(* Logix 5000 project; controller Transcat_L33ER vendor 1 type 14 code 107 rev 32.11; software revision 32.02; part 3 of 4 *)
(* tags used below, declared in another part *)
   AllDevice1stScanDone : BOOL;   // When this bit is set - all devices have been scanned once and bits reset
   AllDeviceEnable : BOOL;   // A bit to enable or disable the running of all devices
   AllReset : BOOL;   // Bit to reset Auto/Man, AutoRun, RecipeRun, TimedRunEnable to 0 from PLC
   alwaysOFF : BOOL;
   AnyAutoRun : BOOL;   // Bit that in on if ANY device is placed into Auto run (to signal pre-start beed)
   AnyAutoRunFlag : BOOL;   // A flag that indicates if any device is in Auto Run (used with pre-start beep logic)
   AnyManRunFlag : BOOL;   // A flag that indicates if any device is in Manual Run (used with pre-start beep logic)
   AnyManualRun : BOOL;   // Bit that in on if ANY device is placed into manual run (to signal pre-start beed)
   Auto_Run_All_Interlock : BOOL;   // Bit to interlock all devices running in Auto
   AutoActive : BOOL;   // Auto mode active
   Beep : BOOL;   // Bit to Activte Beacon Alarm
   Device : Device[20];
   DiscreteTemp : BOOL;   // A temporay boolean to hold positions during PLC transer
   dNum : DINT;   // The index of the current device being processed
   DoseCounter : COUNTER;   // Counts the # of doses since last reset
   DoseCounterReset_HMI : BOOL;   // HMI bit to reset the dose counter
   DoseStart : BOOL;   // Bit to start dosing sequence
   DoseStartOneShot : BOOL;   // One shot to start dosing
   DoseStop : BOOL;   // Bit to stop dosing
   DoseStopOneShot : BOOL;   // one shot to stop dosing
   DoseTarget : REAL;   // Target dose amount
   EstopActive : BOOL;   // E
   EstopFalutResetTOF : TIMER;   // Timer to hold reset bit to allow all drives to reset
   EStopResetPulse : BOOL;   // One-scan pulse used to clear all 14 E-stop interlocks - allows reset of estop interlocks from physical reset button on V
   EStopResetRequired : BOOL;   // Indicates that an estop was actived and it's awaiting reset
   FT103 : BronkhorstFlowMeter;
   FT103B : BronkhorstFlowMeter;
   GF101 : Thayer_WB_Feeder;   // Thayer 1 Tags
   GF101_Write_Acknowledge : ALIAS FOR Thayer1_BS:O.Data[2].5;   // Thayer 1 (GF101) Acknowledge
   GF201 : Thayer_WB_Feeder;   // Thayer 2 Tags
   GF201_Totalizer1 : ALIAS FOR Thayer2Data[9];   // Thayer 2 (GF201) Totalizer 1 in lbs
   GF201_Write_Acknowledge : ALIAS FOR Thayer2_BS:O.Data[2].5;   // Thayer 2 (GF201) Acknowledge
   GF201_Write_Total1Reset : ALIAS FOR Thayer2_BS:O.Data[2].1;   // Thayer 2 (GF1201) Totalizer 1 reset
   HMI_AllReset : BOOL;   // Bit to reset Auto/Man, AutoRun, RecipeRun, TimedRunEnable to 0 from HMI
   HMI_AutoStart : BOOL;   // Starts all devices in AUTO
   HMI_AutoStop : BOOL;   // Stops all devices in AUTO
   HMI_RecipeStart : BOOL;   // Bit to start and stop recipe from HMI
   InitCount : INT;   // Counter to cycle through each device on start-up and reset AutoMan, AutoRun, ManualRun bits
   MX101 : Howes_Mixer;
   MX201 : Howes_Mixer;
   RecipeStart : BOOL;   // Bit to start and stop a recipe execution from PLC logic
   StartBeepTimer : TIMER;   // Timer to sound the beep alarm before starting a device
   TestBit1 : BOOL;   // Just a test bit - does not do anything
   Thayer2ResetTotal1_HMI : BOOL;   // Bit to reset Thayer2 - totalizer 1 from HMI
   VF101 : Acrison_Feeder;   // Medium Feeder Tags
   VF201 : Acrison_Feeder;   // Small Feeder 2 Tags
   VFD_Panel_Safety_Panel_Etop_OK : ALIAS FOR XS26_VFD_Cabinet_Safety_Controller:I1.Data[1].6;
   VFD_Panel_Safety_Remote_Estops_OK : ALIAS FOR XS26_VFD_Cabinet_Safety_Controller:I1.Data[1].7;
(* MainProgram, continued *)

ROUTINE DeviceLogic   (* ladder *)
// Process the logic for each device with index and indirect addressing.
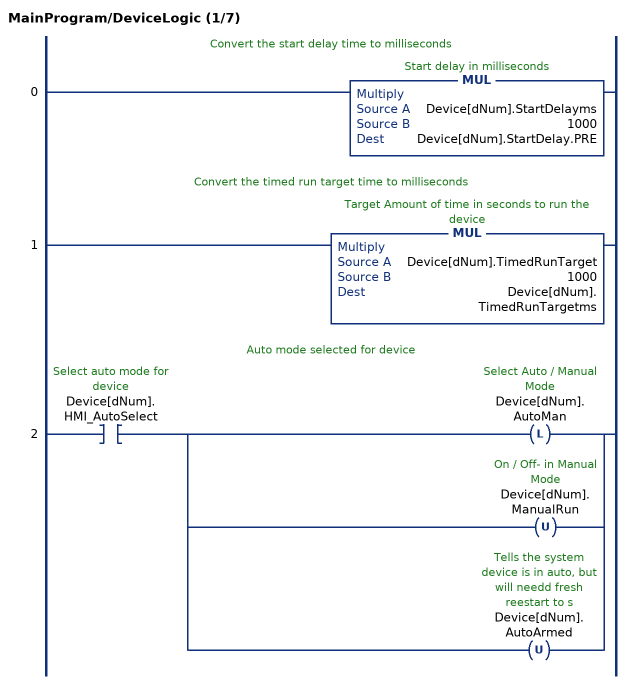
   // Convert the start delay time to milliseconds
   0: MUL(Device[dNum].StartDelayms,1000,Device[dNum].StartDelay.PRE);
   // Convert the timed run target time to milliseconds
   1: MUL(Device[dNum].TimedRunTarget,1000,Device[dNum].TimedRunTargetms);
   // Auto mode selected for device
   2: XIC(Device[dNum].HMI_AutoSelect)[OTL(Device[dNum].AutoMan) ,OTU(Device[dNum].ManualRun) ,OTU(Device[dNum].AutoArmed) ];
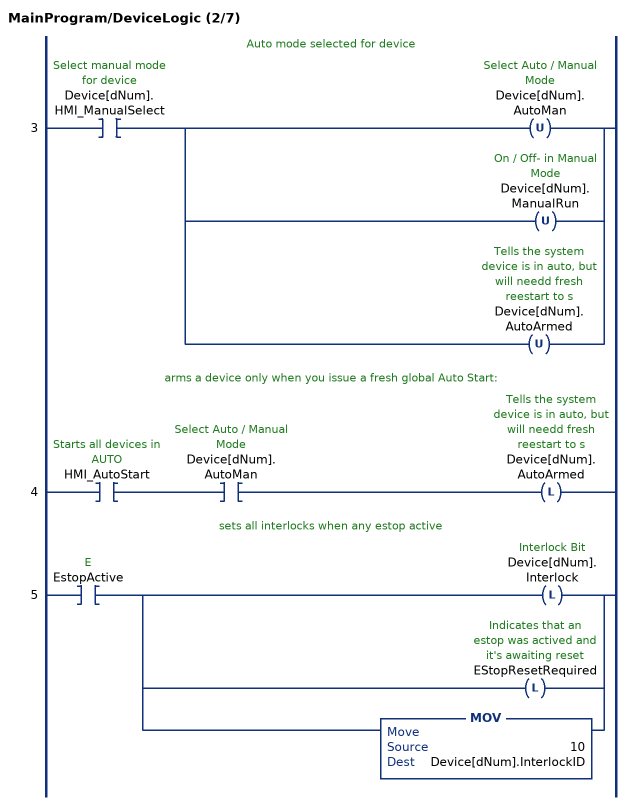
   // Auto mode selected for device
   3: XIC(Device[dNum].HMI_ManualSelect)[OTU(Device[dNum].AutoMan) ,[OTU(Device[dNum].ManualRun) ,OTU(Device[dNum].AutoArmed) ] ];
   // arms a device only when you issue a fresh global Auto Start:
   4: XIC(HMI_AutoStart)XIC(Device[dNum].AutoMan)OTL(Device[dNum].AutoArmed);
   // sets all interlocks when any estop active
   5: XIC(EstopActive)[OTL(Device[dNum].Interlock) ,OTL(EStopResetRequired) ,MOV(10,Device[dNum].InterlockID) ];
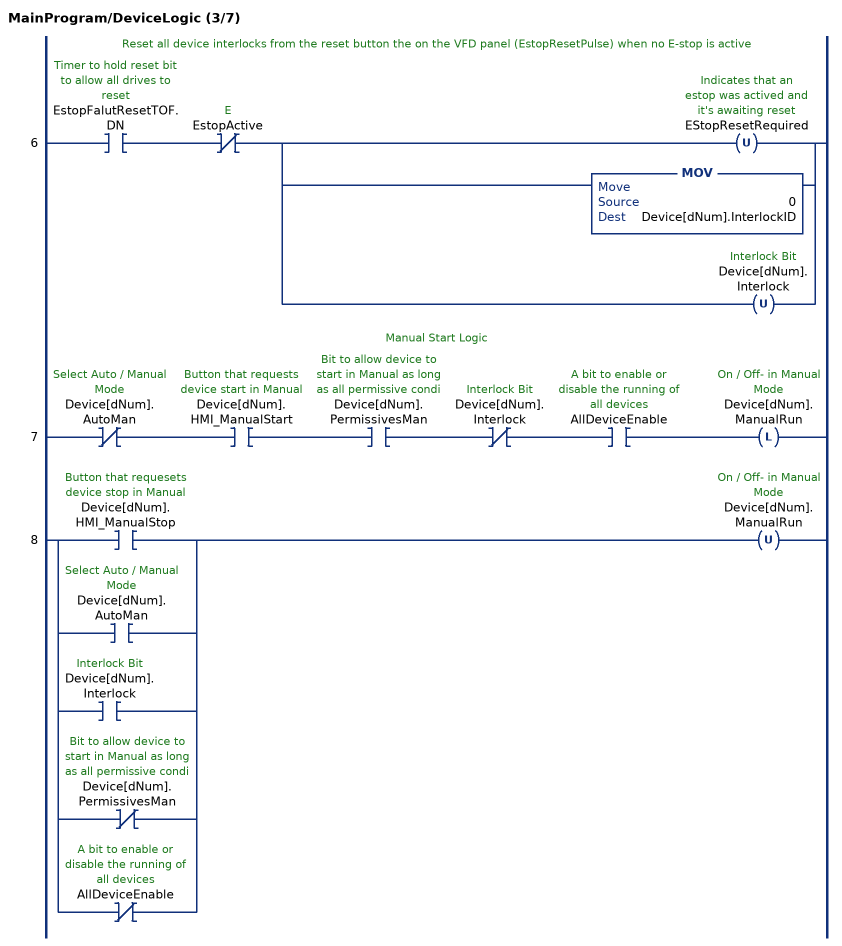
   // Reset all device interlocks from the reset button the on the VFD panel (EstopResetPulse) when no E-stop is active
   6: XIC(EstopFalutResetTOF.DN)XIO(EstopActive)[OTU(EStopResetRequired) ,MOV(0,Device[dNum].InterlockID) ,OTU(Device[dNum].Interlock) ];
   // Manual Start Logic
   7: XIO(Device[dNum].AutoMan)XIC(Device[dNum].HMI_ManualStart)XIC(Device[dNum].PermissivesMan)XIO(Device[dNum].Interlock)XIC(AllDeviceEnable)OTL(Device[dNum].ManualRun);
   8: [XIC(Device[dNum].HMI_ManualStop) ,[XIC(Device[dNum].AutoMan) ,[XIC(Device[dNum].Interlock) ,[XIO(Device[dNum].PermissivesMan) ,XIO(AllDeviceEnable) ] ] ] ]OTU(Device[dNum].ManualRun);
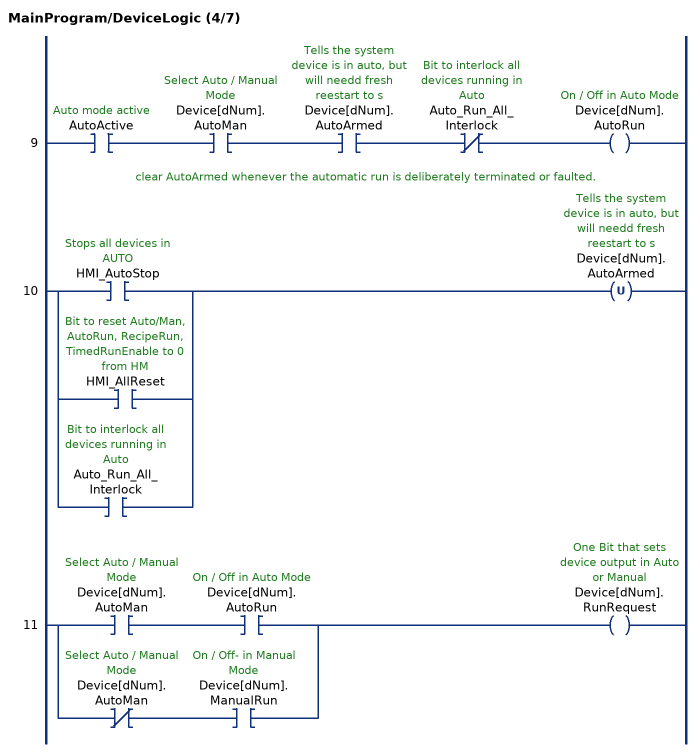
   9: XIC(AutoActive)XIC(Device[dNum].AutoMan)XIC(Device[dNum].AutoArmed)XIO(Auto_Run_All_Interlock)OTE(Device[dNum].AutoRun);
   // clear AutoArmed whenever the automatic run is deliberately terminated or faulted.
   10: [XIC(HMI_AutoStop) ,[XIC(HMI_AllReset) ,XIC(Auto_Run_All_Interlock) ] ]OTU(Device[dNum].AutoArmed);
   11: [XIC(Device[dNum].AutoMan) XIC(Device[dNum].AutoRun) ,XIO(Device[dNum].AutoMan) XIC(Device[dNum].ManualRun) ]OTE(Device[dNum].RunRequest);
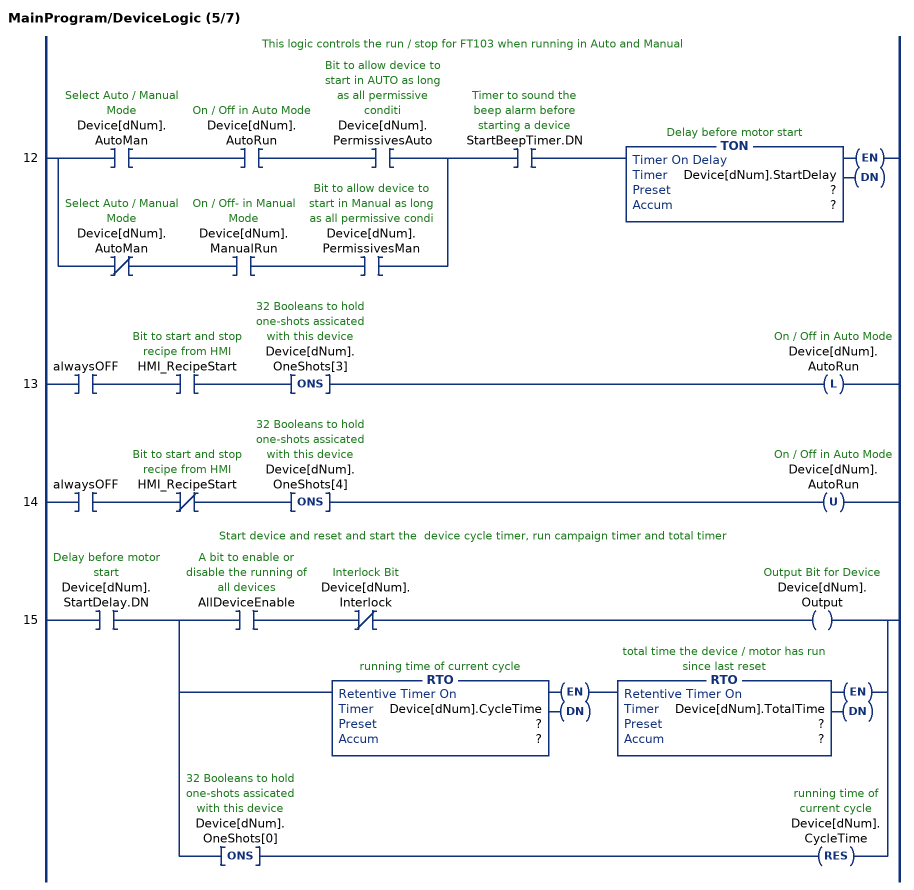
   // This logic controls the run / stop for FT103 when running in Auto and Manual
   12: [XIC(Device[dNum].AutoMan) XIC(Device[dNum].AutoRun) XIC(Device[dNum].PermissivesAuto) ,XIO(Device[dNum].AutoMan) XIC(Device[dNum].ManualRun) XIC(Device[dNum].PermissivesMan) ]XIC(StartBeepTimer.DN)TON(Device[dNum].StartDelay,?,?);
   13: XIC(alwaysOFF)XIC(HMI_RecipeStart)ONS(Device[dNum].OneShots[3])OTL(Device[dNum].AutoRun);
   14: XIC(alwaysOFF)XIO(HMI_RecipeStart)ONS(Device[dNum].OneShots[4])OTU(Device[dNum].AutoRun);
   // Start device and reset and start the  device cycle timer, run campaign timer and total timer
   15: XIC(Device[dNum].StartDelay.DN)[XIC(AllDeviceEnable) XIO(Device[dNum].Interlock) OTE(Device[dNum].Output) ,[RTO(Device[dNum].CycleTime,?,?) RTO(Device[dNum].TotalTime,?,?) ,ONS(Device[dNum].OneShots[0]) RES(Device[dNum].CycleTime) ] ];
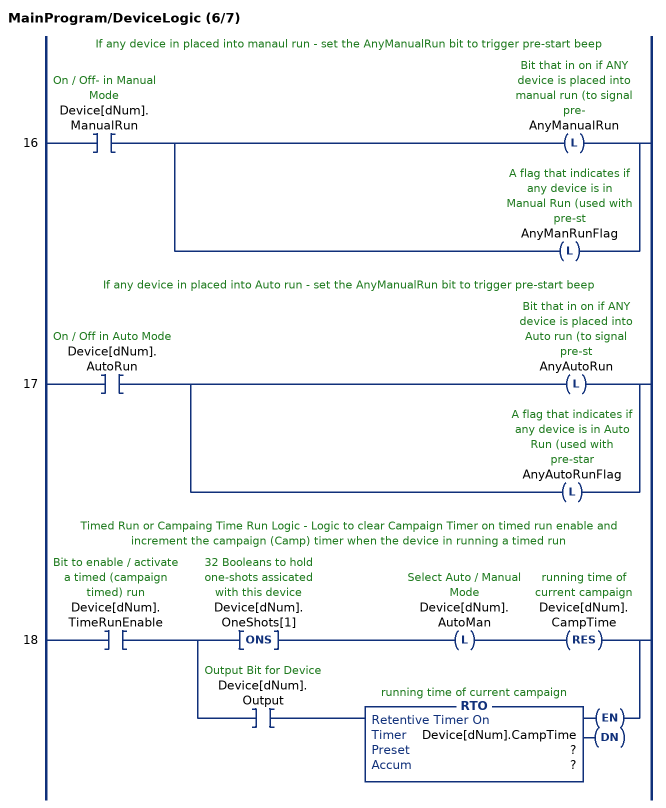
   // If any device in placed into manaul run - set the AnyManualRun bit to trigger pre-start beep
   16: XIC(Device[dNum].ManualRun)[OTL(AnyManualRun) ,OTL(AnyManRunFlag) ];
   // If any device in placed into Auto run - set the AnyManualRun bit to trigger pre-start beep
   17: XIC(Device[dNum].AutoRun)[OTL(AnyAutoRun) ,OTL(AnyAutoRunFlag) ];
   // Timed Run or Campaing Time Run Logic - Logic to clear Campaign Timer on timed run enable and increment the campaign (Camp) timer when the device in running a timed run
   18: XIC(Device[dNum].TimeRunEnable)[ONS(Device[dNum].OneShots[1]) OTL(Device[dNum].AutoMan) RES(Device[dNum].CampTime) ,XIC(Device[dNum].Output) RTO(Device[dNum].CampTime,?,?) ];
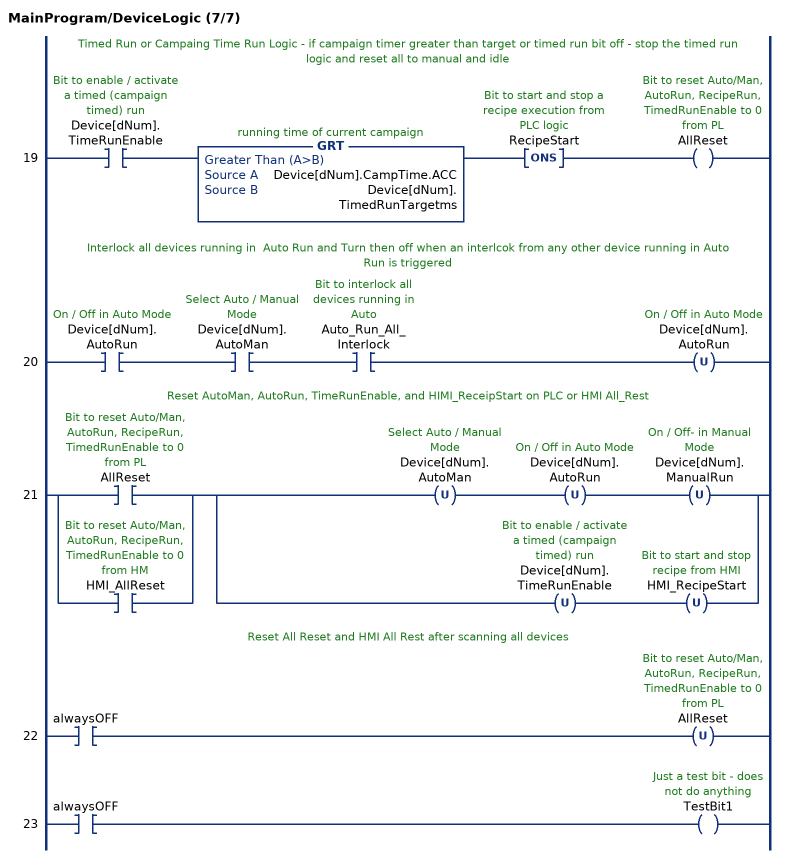
   // Timed Run or Campaing Time Run Logic - if campaign timer greater than target or timed run bit off - stop the timed run logic and reset all to manual and idle
   19: XIC(Device[dNum].TimeRunEnable)GRT(Device[dNum].CampTime.ACC,Device[dNum].TimedRunTargetms)ONS(RecipeStart)OTE(AllReset);
   // Interlock all devices running in  Auto Run and Turn then off when an interlcok from any other device running in Auto Run is triggered
   20: XIC(Device[dNum].AutoRun)XIC(Device[dNum].AutoMan)XIC(Auto_Run_All_Interlock)OTU(Device[dNum].AutoRun);
   // Reset AutoMan, AutoRun, TimeRunEnable, and HIMI_ReceipStart on PLC or HMI All_Rest
   21: [XIC(AllReset) ,XIC(HMI_AllReset) ][OTU(Device[dNum].AutoMan) OTU(Device[dNum].AutoRun) OTU(Device[dNum].ManualRun) ,OTU(Device[dNum].TimeRunEnable) OTU(HMI_RecipeStart) ];
   // Reset All Reset and HMI All Rest after scanning all devices
   22: XIC(alwaysOFF)OTU(AllReset);
   23: XIC(alwaysOFF)OTE(TestBit1);
END_ROUTINE

ROUTINE DeviceManager   (* ladder *)
// Loop through all devices each scan
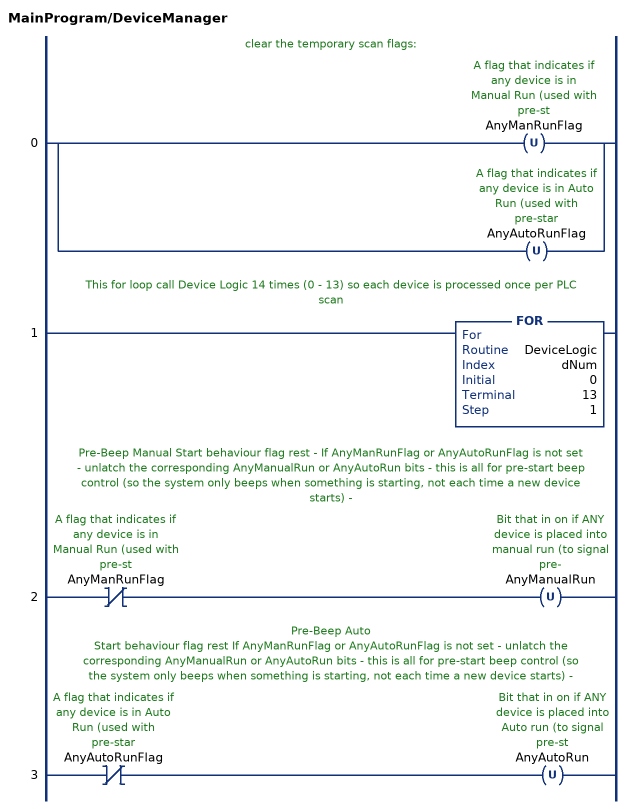
   // clear the temporary scan flags:
   0: [OTU(AnyManRunFlag) ,OTU(AnyAutoRunFlag) ];
   // This for loop call Device Logic 14 times (0 - 13) so each device is processed once per PLC scan
   1: FOR(DeviceLogic,dNum,0,13,1);
   // Pre-Beep Manual Start behaviour flag rest - If AnyManRunFlag or AnyAutoRunFlag is not set - unlatch the corresponding AnyManualRun or AnyAutoRun bits - this is all for pre-start beep control (so the system only beeps when something is starting, not each time a new device starts) -
   2: XIO(AnyManRunFlag)OTU(AnyManualRun);
   // Pre-Beep Auto
   //  Start behaviour flag rest If AnyManRunFlag or AnyAutoRunFlag is not set - unlatch the corresponding AnyManualRun or AnyAutoRun bits - this is all for pre-start beep control (so the system only beeps when something is starting, not each time a new device starts) -
   3: XIO(AnyAutoRunFlag)OTU(AnyAutoRun);
END_ROUTINE

ROUTINE GF201Dose   (* ladder *)
// Logic to Dose a specific amount from GF201 - Thayer 2
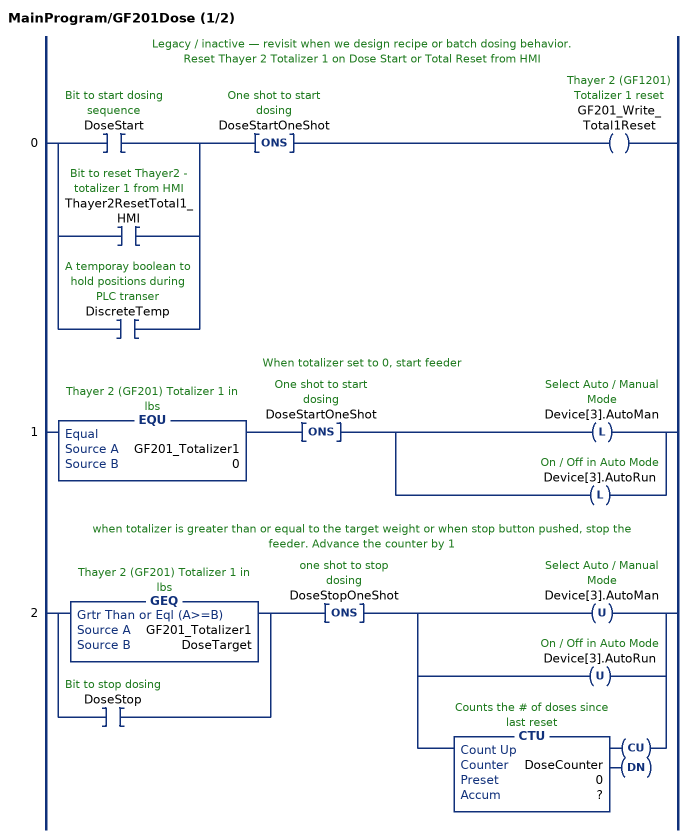
   // Legacy / inactive — revisit when we design recipe or batch dosing behavior.
   // Reset Thayer 2 Totalizer 1 on Dose Start or Total Reset from HMI
   0: [XIC(DoseStart) ,[XIC(Thayer2ResetTotal1_HMI) ,XIC(DiscreteTemp) ] ]ONS(DoseStartOneShot)OTE(GF201_Write_Total1Reset);
   // When totalizer set to 0, start feeder
   1: EQU(GF201_Totalizer1,0)ONS(DoseStartOneShot)[OTL(Device[3].AutoMan) ,OTL(Device[3].AutoRun) ];
   // when totalizer is greater than or equal to the target weight or when stop button pushed, stop the feeder. Advance the counter by 1
   2: [GEQ(GF201_Totalizer1,DoseTarget) ,XIC(DoseStop) ]ONS(DoseStopOneShot)[OTU(Device[3].AutoMan) ,[OTU(Device[3].AutoRun) ,CTU(DoseCounter,?,?) ] ];
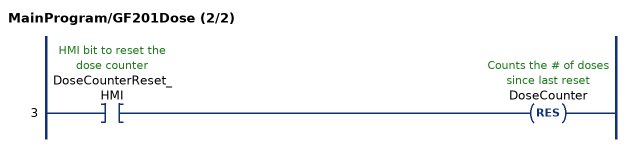
   3: XIC(DoseCounterReset_HMI)RES(DoseCounter);
END_ROUTINE

ROUTINE Initialize   (* ladder *)
// Reset controls and any other initialization required
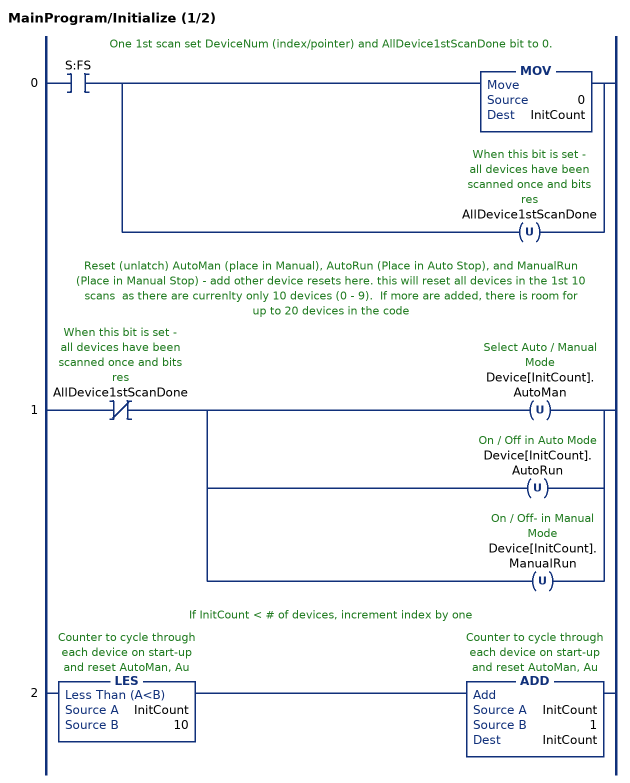
   // One 1st scan set DeviceNum (index/pointer) and AllDevice1stScanDone bit to 0.
   0: XIC(S:FS)[MOV(0,InitCount) ,OTU(AllDevice1stScanDone) ];
   // Reset (unlatch) AutoMan (place in Manual), AutoRun (Place in Auto Stop), and ManualRun (Place in Manual Stop) - add other device resets here. this will reset all devices in the 1st 10 scans  as there are currenlty only 10 devices (0 - 9).  If more are added, there is room for up to 20 devices in the code
   1: XIO(AllDevice1stScanDone)[OTU(Device[InitCount].AutoMan) ,[OTU(Device[InitCount].AutoRun) ,OTU(Device[InitCount].ManualRun) ] ];
   // If InitCount < # of devices, increment index by one
   2: LES(InitCount,10)ADD(InitCount,1,InitCount);
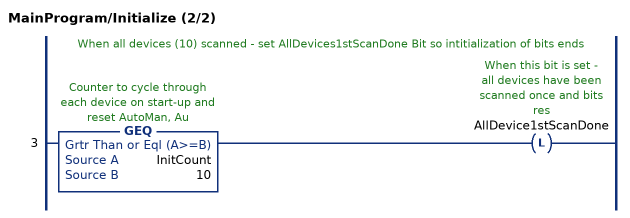
   // When all devices (10) scanned - set AllDevices1stScanDone Bit so intitialization of bits ends
   3: GEQ(InitCount,10)OTL(AllDevice1stScanDone);
END_ROUTINE

ROUTINE InterlockLogic   (* ladder *)
// All interlock logic is handled here
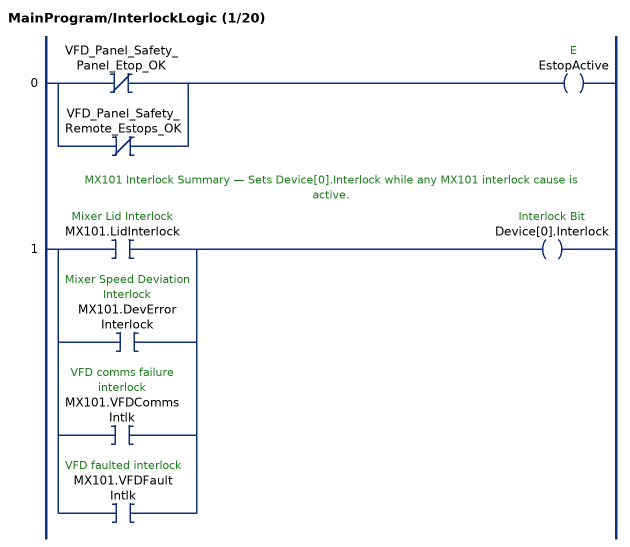
   0: [XIO(VFD_Panel_Safety_Panel_Etop_OK) ,XIO(VFD_Panel_Safety_Remote_Estops_OK) ]OTE(EstopActive);
   // MX101 Interlock Summary — Sets Device[0].Interlock while any MX101 interlock cause is active.
   1: [XIC(MX101.LidInterlock) ,XIC(MX101.DevErrorInterlock) ,XIC(MX101.VFDCommsIntlk) ,XIC(MX101.VFDFaultIntlk) ]OTE(Device[0].Interlock);
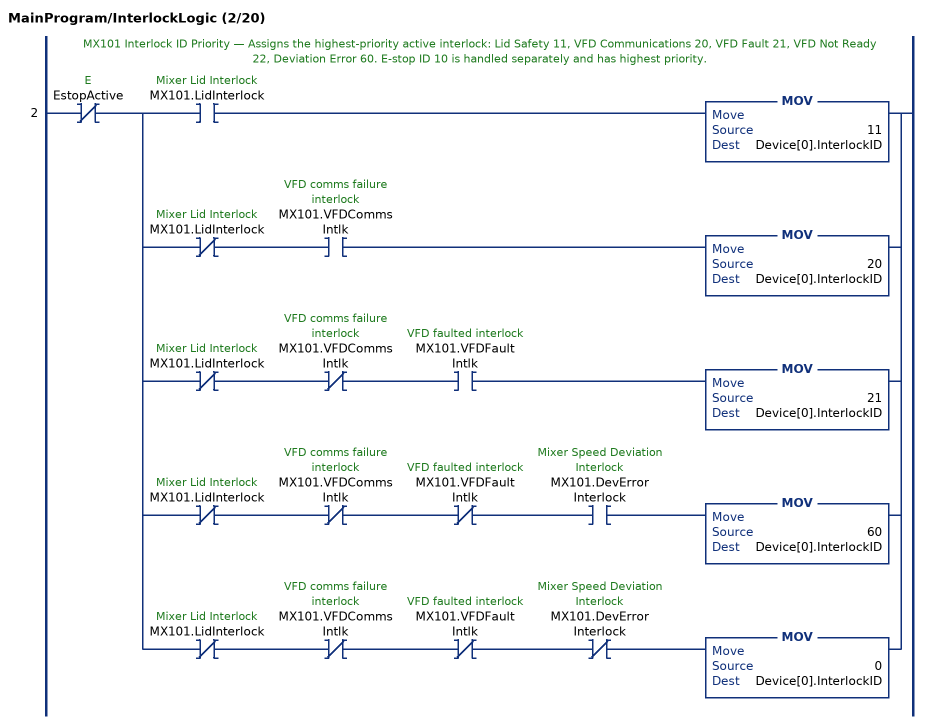
   // MX101 Interlock ID Priority — Assigns the highest-priority active interlock: Lid Safety 11, VFD Communications 20, VFD Fault 21, VFD Not Ready 22, Deviation Error 60. E-stop ID 10 is handled separately and has highest priority.
   2: XIO(EstopActive)[XIC(MX101.LidInterlock) MOV(11,Device[0].InterlockID) ,XIO(MX101.LidInterlock) XIC(MX101.VFDCommsIntlk) MOV(20,Device[0].InterlockID) ,XIO(MX101.LidInterlock) XIO(MX101.VFDCommsIntlk) XIC(MX101.VFDFaultIntlk) MOV(21,Device[0].InterlockID) ,XIO(MX101.LidInterlock) XIO(MX101.VFDCommsIntlk) XIO(MX101.VFDFaultIntlk) XIC(MX101.DevErrorInterlock) MOV(60,Device[0].InterlockID) ,XIO(MX101.LidInterlock) XIO(MX101.VFDCommsIntlk) XIO(MX101.VFDFaultIntlk) XIO(MX101.DevErrorInterlock) MOV(0,Device[0].InterlockID) ];
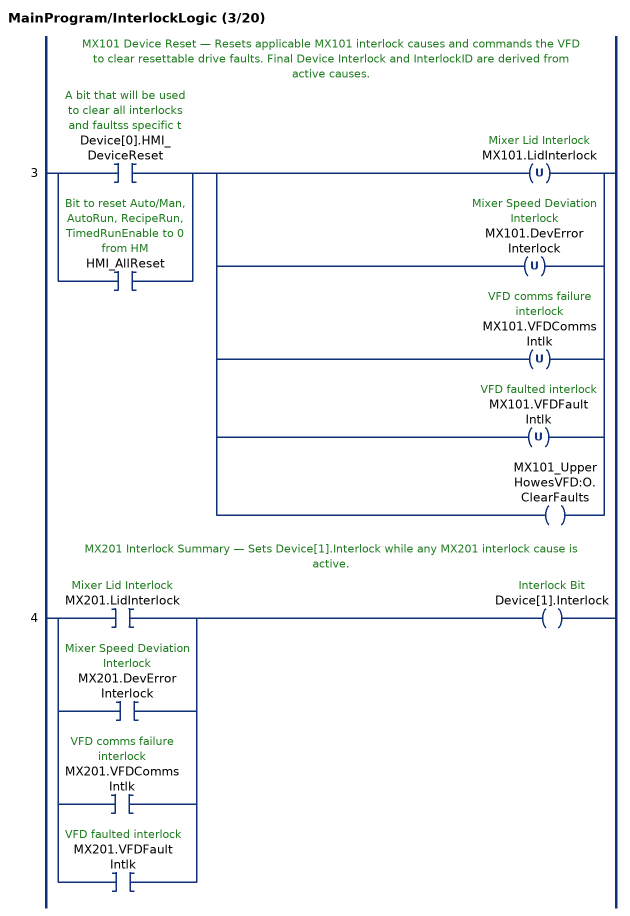
   // MX101 Device Reset — Resets applicable MX101 interlock causes and commands the VFD to clear resettable drive faults. Final Device Interlock and InterlockID are derived from active causes.
   3: [XIC(Device[0].HMI_DeviceReset) ,XIC(HMI_AllReset) ][OTU(MX101.LidInterlock) ,OTU(MX101.DevErrorInterlock) ,OTU(MX101.VFDCommsIntlk) ,OTU(MX101.VFDFaultIntlk) ,OTE(MX101_UpperHowesVFD:O.ClearFaults) ];
   // MX201 Interlock Summary — Sets Device[1].Interlock while any MX201 interlock cause is active.
   4: [XIC(MX201.LidInterlock) ,XIC(MX201.DevErrorInterlock) ,XIC(MX201.VFDCommsIntlk) ,XIC(MX201.VFDFaultIntlk) ]OTE(Device[1].Interlock);
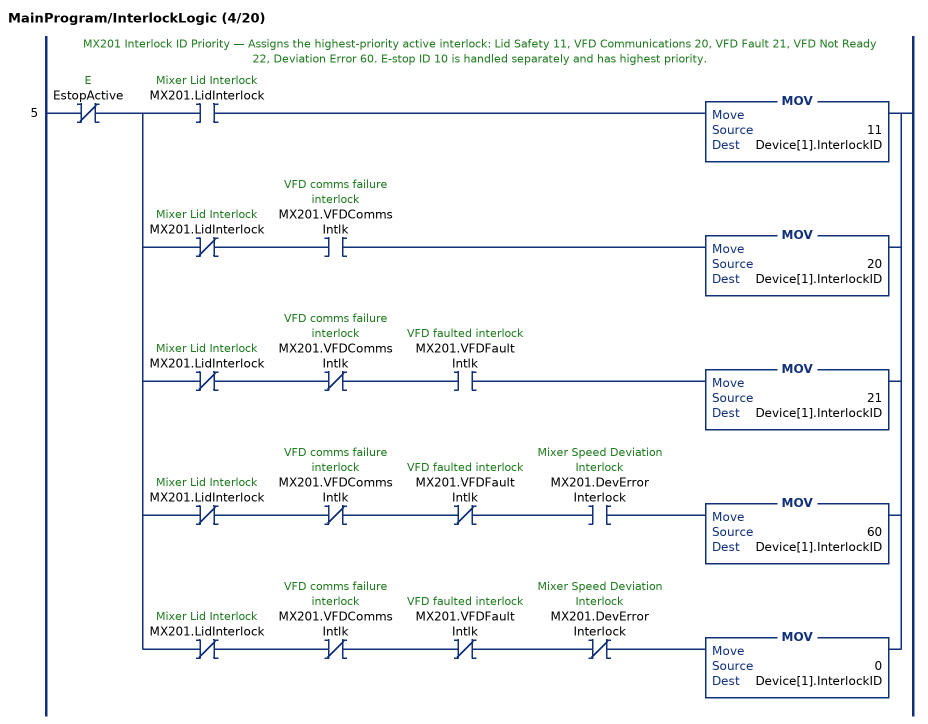
   // MX201 Interlock ID Priority — Assigns the highest-priority active interlock: Lid Safety 11, VFD Communications 20, VFD Fault 21, VFD Not Ready 22, Deviation Error 60. E-stop ID 10 is handled separately and has highest priority.
   5: XIO(EstopActive)[XIC(MX201.LidInterlock) MOV(11,Device[1].InterlockID) ,XIO(MX201.LidInterlock) XIC(MX201.VFDCommsIntlk) MOV(20,Device[1].InterlockID) ,XIO(MX201.LidInterlock) XIO(MX201.VFDCommsIntlk) XIC(MX201.VFDFaultIntlk) MOV(21,Device[1].InterlockID) ,XIO(MX201.LidInterlock) XIO(MX201.VFDCommsIntlk) XIO(MX201.VFDFaultIntlk) XIC(MX201.DevErrorInterlock) MOV(60,Device[1].InterlockID) ,XIO(MX201.LidInterlock) XIO(MX201.VFDCommsIntlk) XIO(MX201.VFDFaultIntlk) XIO(MX201.DevErrorInterlock) MOV(0,Device[1].InterlockID) ];
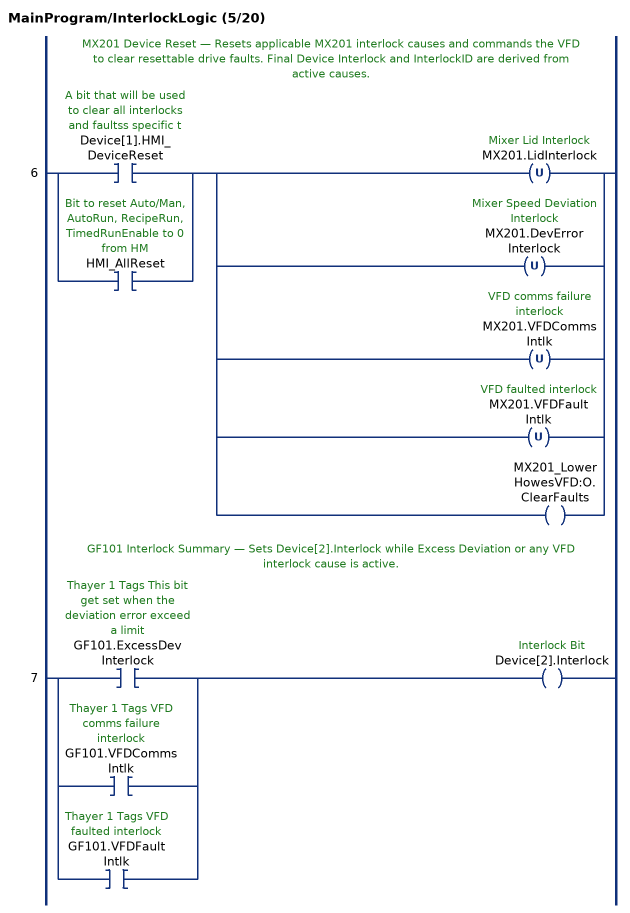
   // MX201 Device Reset — Resets applicable MX201 interlock causes and commands the VFD to clear resettable drive faults. Final Device Interlock and InterlockID are derived from active causes.
   6: [XIC(Device[1].HMI_DeviceReset) ,XIC(HMI_AllReset) ][OTU(MX201.LidInterlock) ,OTU(MX201.DevErrorInterlock) ,OTU(MX201.VFDCommsIntlk) ,OTU(MX201.VFDFaultIntlk) ,OTE(MX201_LowerHowesVFD:O.ClearFaults) ];
   // GF101 Interlock Summary — Sets Device[2].Interlock while Excess Deviation or any VFD interlock cause is active.
   7: [XIC(GF101.ExcessDevInterlock) ,XIC(GF101.VFDCommsIntlk) ,XIC(GF101.VFDFaultIntlk) ]OTE(Device[2].Interlock);
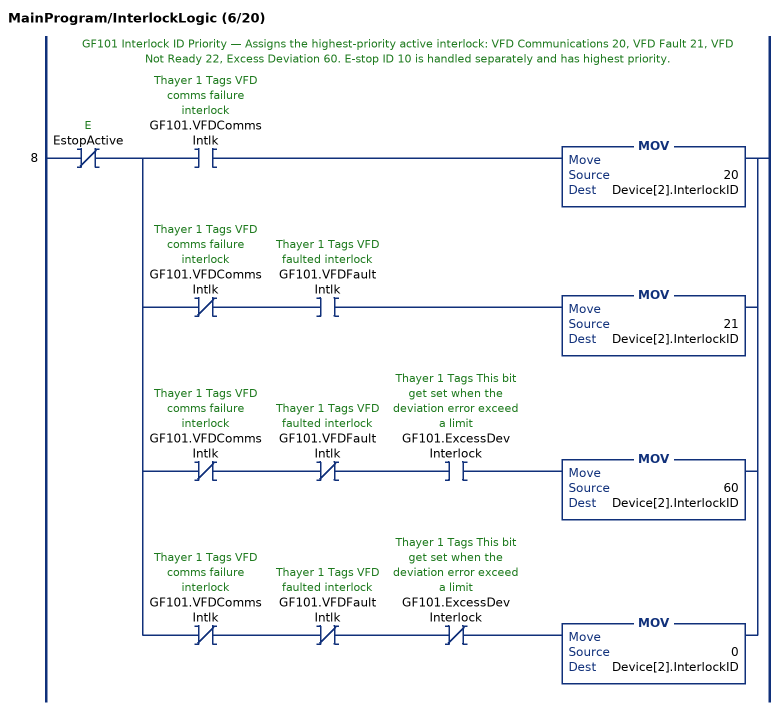
   // GF101 Interlock ID Priority — Assigns the highest-priority active interlock: VFD Communications 20, VFD Fault 21, VFD Not Ready 22, Excess Deviation 60. E-stop ID 10 is handled separately and has highest priority.
   8: XIO(EstopActive)[XIC(GF101.VFDCommsIntlk) MOV(20,Device[2].InterlockID) ,XIO(GF101.VFDCommsIntlk) XIC(GF101.VFDFaultIntlk) MOV(21,Device[2].InterlockID) ,XIO(GF101.VFDCommsIntlk) XIO(GF101.VFDFaultIntlk) XIC(GF101.ExcessDevInterlock) MOV(60,Device[2].InterlockID) ,XIO(GF101.VFDCommsIntlk) XIO(GF101.VFDFaultIntlk) XIO(GF101.ExcessDevInterlock) MOV(0,Device[2].InterlockID) ];
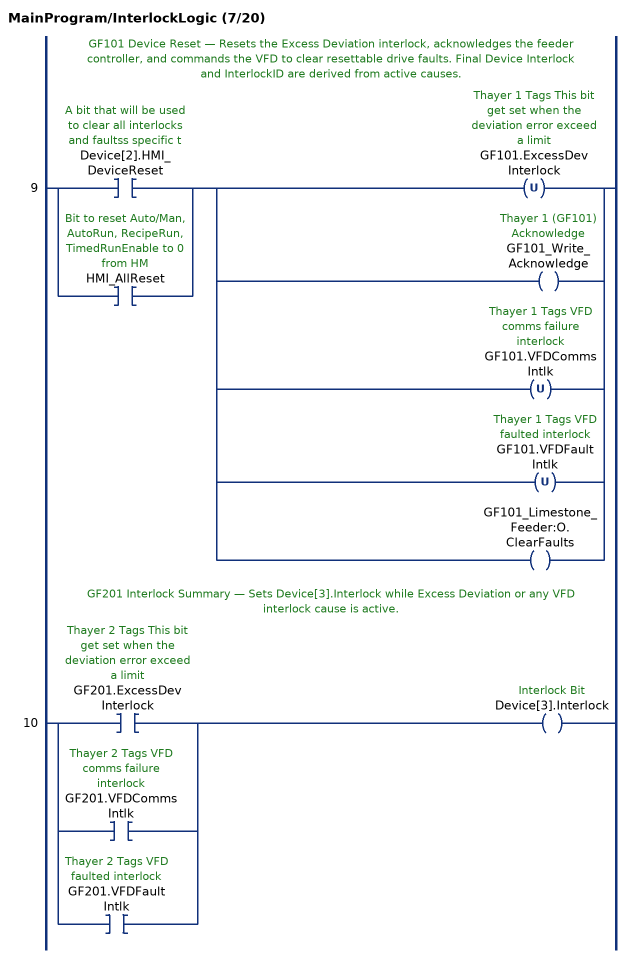
   // GF101 Device Reset — Resets the Excess Deviation interlock, acknowledges the feeder controller, and commands the VFD to clear resettable drive faults. Final Device Interlock and InterlockID are derived from active causes.
   9: [XIC(Device[2].HMI_DeviceReset) ,XIC(HMI_AllReset) ][OTU(GF101.ExcessDevInterlock) ,OTE(GF101_Write_Acknowledge) ,OTU(GF101.VFDCommsIntlk) ,OTU(GF101.VFDFaultIntlk) ,OTE(GF101_Limestone_Feeder:O.ClearFaults) ];
   // GF201 Interlock Summary — Sets Device[3].Interlock while Excess Deviation or any VFD interlock cause is active.
   10: [XIC(GF201.ExcessDevInterlock) ,XIC(GF201.VFDCommsIntlk) ,XIC(GF201.VFDFaultIntlk) ]OTE(Device[3].Interlock);
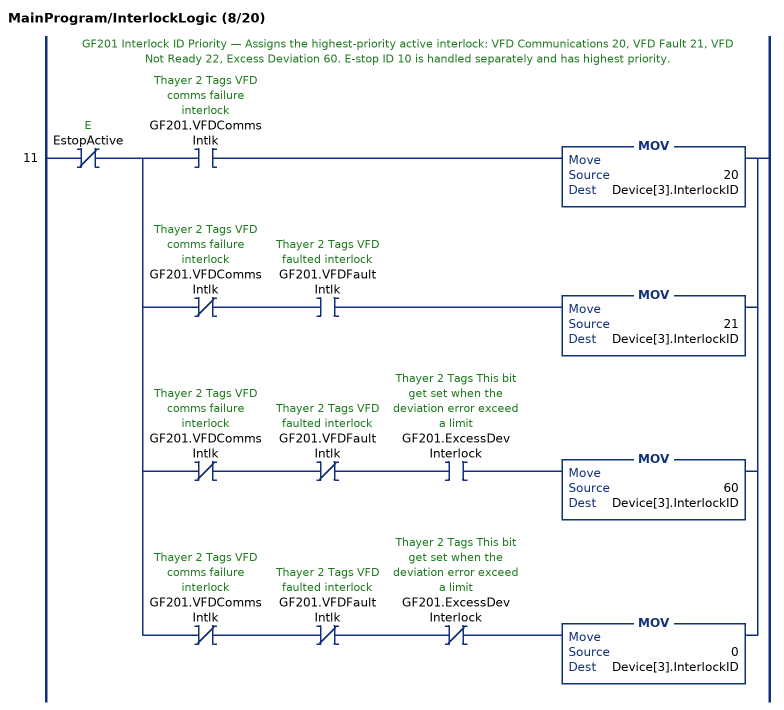
   // GF201 Interlock ID Priority — Assigns the highest-priority active interlock: VFD Communications 20, VFD Fault 21, VFD Not Ready 22, Excess Deviation 60. E-stop ID 10 is handled separately and has highest priority.
   11: XIO(EstopActive)[XIC(GF201.VFDCommsIntlk) MOV(20,Device[3].InterlockID) ,XIO(GF201.VFDCommsIntlk) XIC(GF201.VFDFaultIntlk) MOV(21,Device[3].InterlockID) ,XIO(GF201.VFDCommsIntlk) XIO(GF201.VFDFaultIntlk) XIC(GF201.ExcessDevInterlock) MOV(60,Device[3].InterlockID) ,XIO(GF201.VFDCommsIntlk) XIO(GF201.VFDFaultIntlk) XIO(GF201.ExcessDevInterlock) MOV(0,Device[3].InterlockID) ];
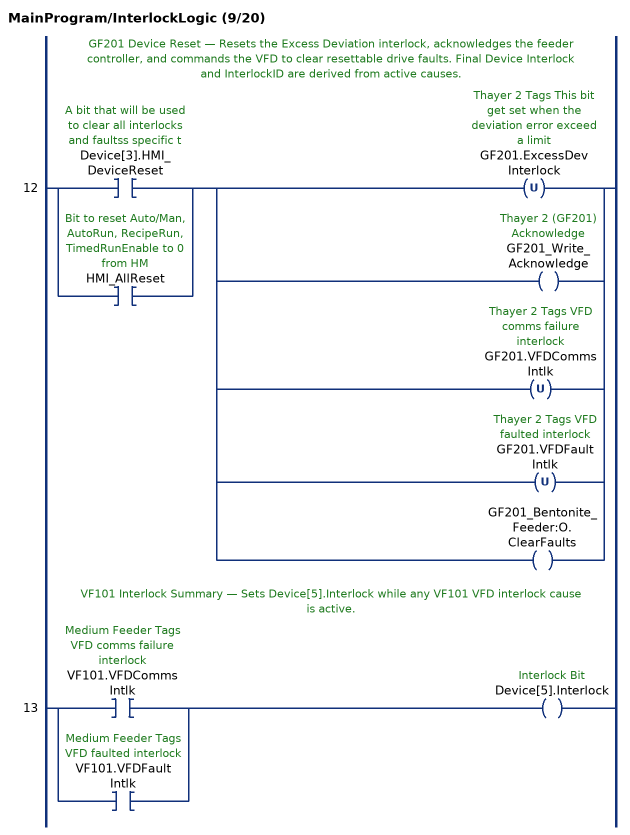
   // GF201 Device Reset — Resets the Excess Deviation interlock, acknowledges the feeder controller, and commands the VFD to clear resettable drive faults. Final Device Interlock and InterlockID are derived from active causes.
   12: [XIC(Device[3].HMI_DeviceReset) ,XIC(HMI_AllReset) ][OTU(GF201.ExcessDevInterlock) ,OTE(GF201_Write_Acknowledge) ,OTU(GF201.VFDCommsIntlk) ,OTU(GF201.VFDFaultIntlk) ,OTE(GF201_Bentonite_Feeder:O.ClearFaults) ];
   // VF101 Interlock Summary — Sets Device[5].Interlock while any VF101 VFD interlock cause is active.
   13: [XIC(VF101.VFDCommsIntlk) ,XIC(VF101.VFDFaultIntlk) ]OTE(Device[5].Interlock);
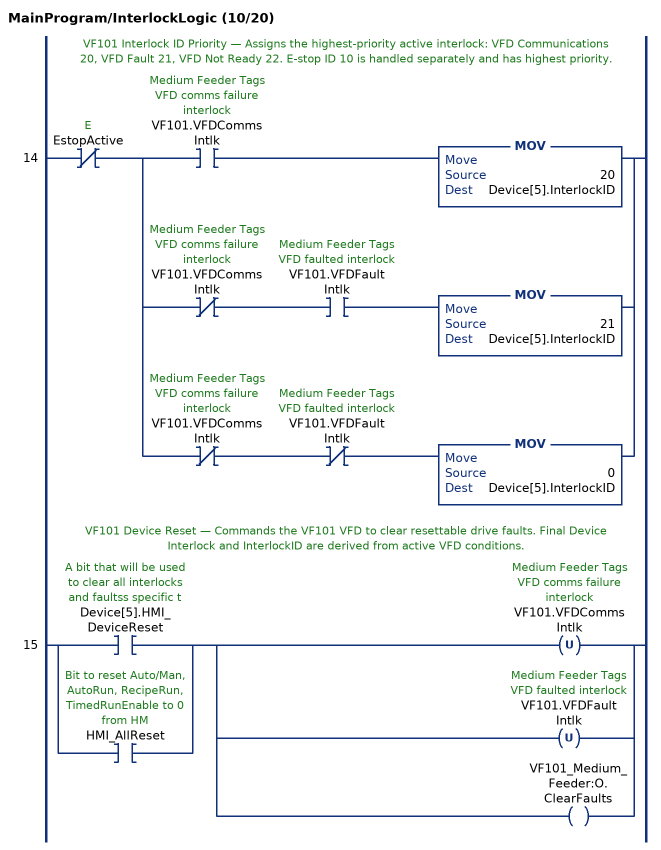
   // VF101 Interlock ID Priority — Assigns the highest-priority active interlock: VFD Communications 20, VFD Fault 21, VFD Not Ready 22. E-stop ID 10 is handled separately and has highest priority.
   14: XIO(EstopActive)[XIC(VF101.VFDCommsIntlk) MOV(20,Device[5].InterlockID) ,XIO(VF101.VFDCommsIntlk) XIC(VF101.VFDFaultIntlk) MOV(21,Device[5].InterlockID) ,XIO(VF101.VFDCommsIntlk) XIO(VF101.VFDFaultIntlk) MOV(0,Device[5].InterlockID) ];
   // VF101 Device Reset — Commands the VF101 VFD to clear resettable drive faults. Final Device Interlock and InterlockID are derived from active VFD conditions.
   15: [XIC(Device[5].HMI_DeviceReset) ,XIC(HMI_AllReset) ][OTU(VF101.VFDCommsIntlk) ,OTU(VF101.VFDFaultIntlk) ,OTE(VF101_Medium_Feeder:O.ClearFaults) ];
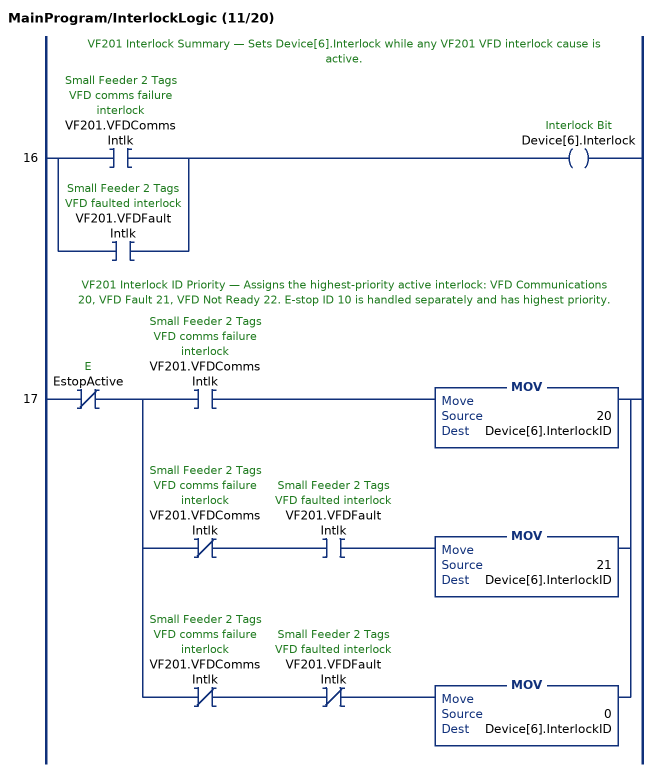
   // VF201 Interlock Summary — Sets Device[6].Interlock while any VF201 VFD interlock cause is active.
   16: [XIC(VF201.VFDCommsIntlk) ,XIC(VF201.VFDFaultIntlk) ]OTE(Device[6].Interlock);
   // VF201 Interlock ID Priority — Assigns the highest-priority active interlock: VFD Communications 20, VFD Fault 21, VFD Not Ready 22. E-stop ID 10 is handled separately and has highest priority.
   17: XIO(EstopActive)[XIC(VF201.VFDCommsIntlk) MOV(20,Device[6].InterlockID) ,XIO(VF201.VFDCommsIntlk) XIC(VF201.VFDFaultIntlk) MOV(21,Device[6].InterlockID) ,XIO(VF201.VFDCommsIntlk) XIO(VF201.VFDFaultIntlk) MOV(0,Device[6].InterlockID) ];
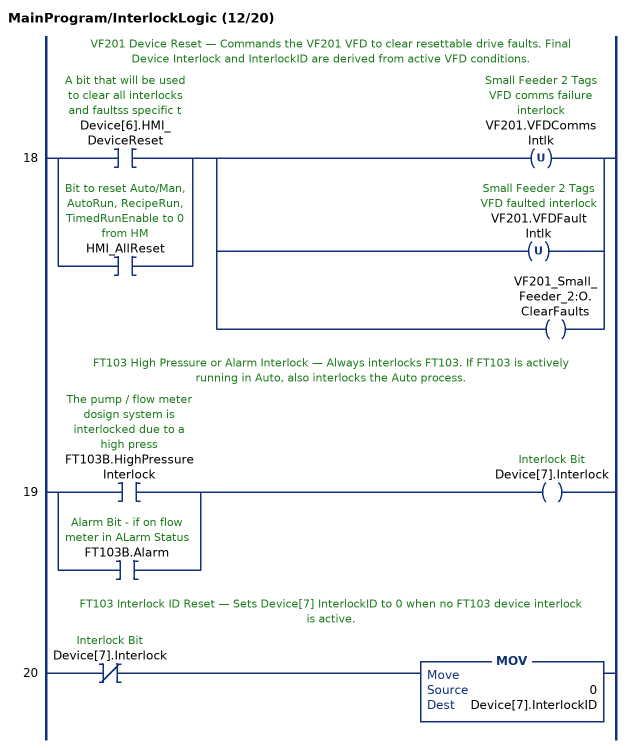
   // VF201 Device Reset — Commands the VF201 VFD to clear resettable drive faults. Final Device Interlock and InterlockID are derived from active VFD conditions.
   18: [XIC(Device[6].HMI_DeviceReset) ,XIC(HMI_AllReset) ][OTU(VF201.VFDCommsIntlk) ,OTU(VF201.VFDFaultIntlk) ,OTE(VF201_Small_Feeder_2:O.ClearFaults) ];
   // FT103 High Pressure or Alarm Interlock — Always interlocks FT103. If FT103 is actively running in Auto, also interlocks the Auto process.
   19: [XIC(FT103B.HighPressureInterlock) ,XIC(FT103B.Alarm) ]OTE(Device[7].Interlock);
   // FT103 Interlock ID Reset — Sets Device[7] InterlockID to 0 when no FT103 device interlock is active.
   20: XIO(Device[7].Interlock)MOV(0,Device[7].InterlockID);
